// Mitsubishi GX Works2 project: gd   PLC: Q03UDV

PROGRAM MAIN
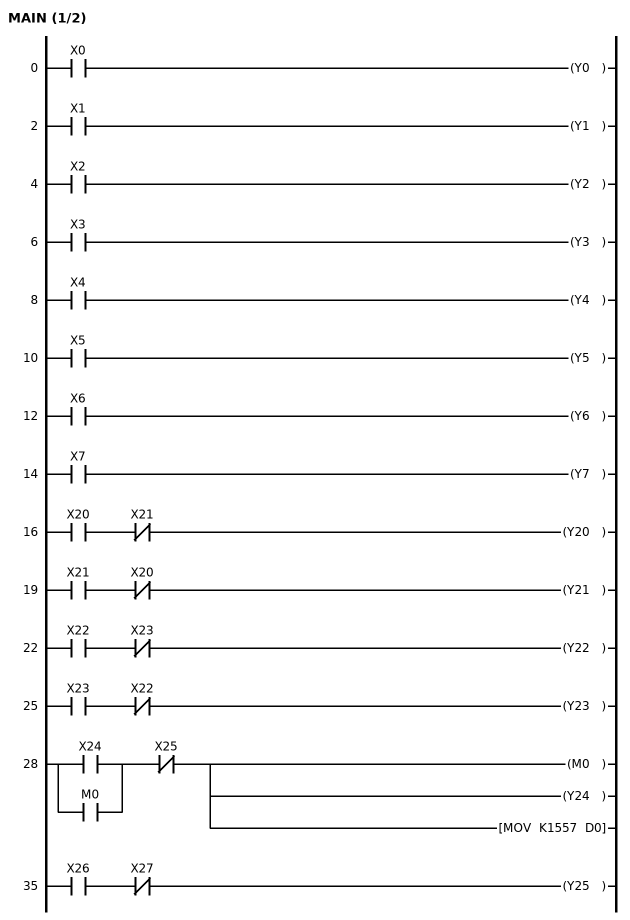
0     LD      X0
      OUT     Y0
2     LD      X1
      OUT     Y1
4     LD      X2
      OUT     Y2
6     LD      X3
      OUT     Y3
8     LD      X4
      OUT     Y4
10    LD      X5
      OUT     Y5
12    LD      X6
      OUT     Y6
14    LD      X7
      OUT     Y7
16    LD      X20
      ANI     X21
      OUT     Y20
19    LD      X21
      ANI     X20
      OUT     Y21
22    LD      X22
      ANI     X23
      OUT     Y22
25    LD      X23
      ANI     X22
      OUT     Y23
28    LD      X24
      OR      M0
      ANI     X25
      OUT     M0
      OUT     Y24
      MOV     K1557 D0
35    LD      X26
      ANI     X27
      OUT     Y25
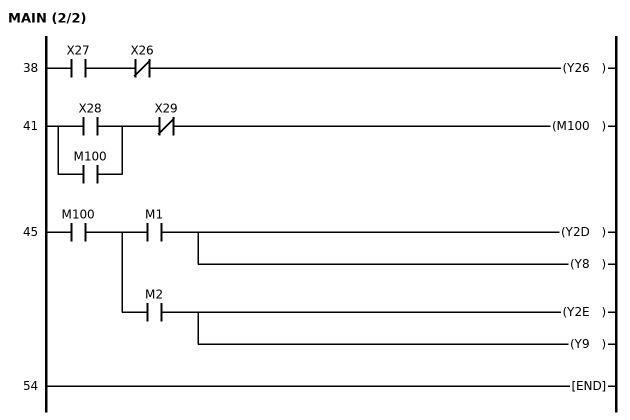
38    LD      X27
      ANI     X26
      OUT     Y26
41    LD      X28
      OR      M100
      ANI     X29
      OUT     M100
45    LD      M100
      MPS
      AND     M1
      OUT     Y2D
      OUT     Y8
      MPP
      AND     M2
      OUT     Y2E
      OUT     Y9
54    END
END_PROGRAM
